# EPICS autosave request: iocBoot/iocpdu/auto_settings.req
file "netbooter5_settings.req" P=$(P),R=pdu5_1:
